PROGRAM MAIN
VAR
END_VAR

END_PROGRAM

(* stored: Version 1.1.0.1
   POU MAIN: Id {753650ed-5d0e-43b3-92c0-79c094ab6917} *)
